(* CoDeSys 2.3.9.50 project: A_I_finale.pro *)
(* Libraries: STANDARD.LIB 5.6.98 12:03:02, Iecsfc.lib 12.5.98 12:03:00 *)

(* Task configuration *)
TASK Standard (PRIORITY := 0, INTERVAL := T#10ms);
	MAIN
END_TASK

(* POU MAIN, SFC *)
PROGRAM MAIN
VAR
	Presenza_pezzo								AT %IX0.0:BOOL;
	Colore_giostra								AT %IX0.1:BOOL;
	Pistone_avanti								AT %IX0.2:BOOL;
	Trapano_alto									AT %IX0.3:BOOL;
	Pistone_indietro								AT %IX0.4:BOOL;
	Trapano_basso								AT %IX0.5:BOOL;
	Fine_corsa_nastro								AT %IX0.6:BOOL;
	Tastatore_alto_altezza							AT %IX0.7:BOOL;


	Scarto_giostra_avanti_post_6					AT %IX1.0:BOOL;
	Scarto_giostra_indietro_post_6					AT %IX1.1:BOOL;
	Presenza_pezzo_baia							AT %IX1.2:BOOL;
	Tastatore_basso_altezza						AT %IX1.3:BOOL;
	Pennarello_alto								AT %IX1.4:BOOL;
	Pennarello_basso								AT %IX1.5:BOOL;
	Scarto_giostra_avanti_post_7					AT %IX1.6:BOOL;
	Scarto_giostra_indietro_post_7					AT %IX1.7:BOOL;


	Giostra_in_movimento							AT%IX2.0:BOOL;
	Sensore_vacuostato							AT%IX2.5:BOOL;
	Fine_corsa_braccio_magazzino					AT%IX2.6:BOOL;
	Presenza_pezzo_magazzino_B4					AT%IX2.7:BOOL;


	Pistone_indietro_1B2							AT%IX3.0:BOOL;
	Pistone_avanti_1B1							AT%IX3.1:BOOL;


	Fine_corsa_braccio_nastro						AT%IX4.1:BOOL;


(* ____ USCITE FISICHE____*)

	nastro  										AT %QX0.0:BOOL;
	pistone_giostra_post_6  						AT %QX0.1:BOOL;
	pistone_nastro		         						AT %QX0.2:BOOL;
	pennarello_down	     	    						AT %QX0.3:BOOL;
	movimento_giostra_1_posto  					AT %QX0.4:BOOL;
	pistone_giostra_post_7  						AT %QX0.5:BOOL;
	trapano_down								AT %QX0.6:BOOL;
	trapano_ON									AT %QX0.7:BOOL;

	tastatore_down								AT %QX1.0:BOOL;

	pistone_orizzontale							AT %QX2.1:BOOL;
	vacuostato									AT %QX2.2:BOOL;
	soffio_aria_ventosa							AT %QX2.3:BOOL;
	braccio_pneumatico_indietro					AT %QX2.4:BOOL;
	braccio_pneumatico_avanti						AT %QX2.5:BOOL;



(* ____ TIMER E CONTATORI IMPLEMENTATI____*)

(* ____ VARIABILI DI APPOGGIO VIRTUALI____*)

	attesa_magazzino: BOOL;
	pezzo_pronto_per_braccio: BOOL;
	pezzo_nel_braccio: BOOL;
	pezzo_pres: BOOL;
	riconoscimento_colore: BOOL;
	t_soffio: TON;
	attesa_secondi: BOOL;

	start:BOOL;
	emergenza:BOOL;
	accensione_pistone:BOOL;
	prova: tempo_3s;
	prova_2: tempo_3s;
	led_bottone: BOOL;
	lancio: BOOL;
	prov: TON;
	passaggio:BOOL;
	controllo_a_campione: CTU;
	pezzo_ok: BOOL;
	reset_cont: BOOL;
	contatore:BOOL;
END_VAR
VAR (* helpers for the ST form of the networks *)
	_p1 : BOOL;
	_p2 : BOOL;
END_VAR
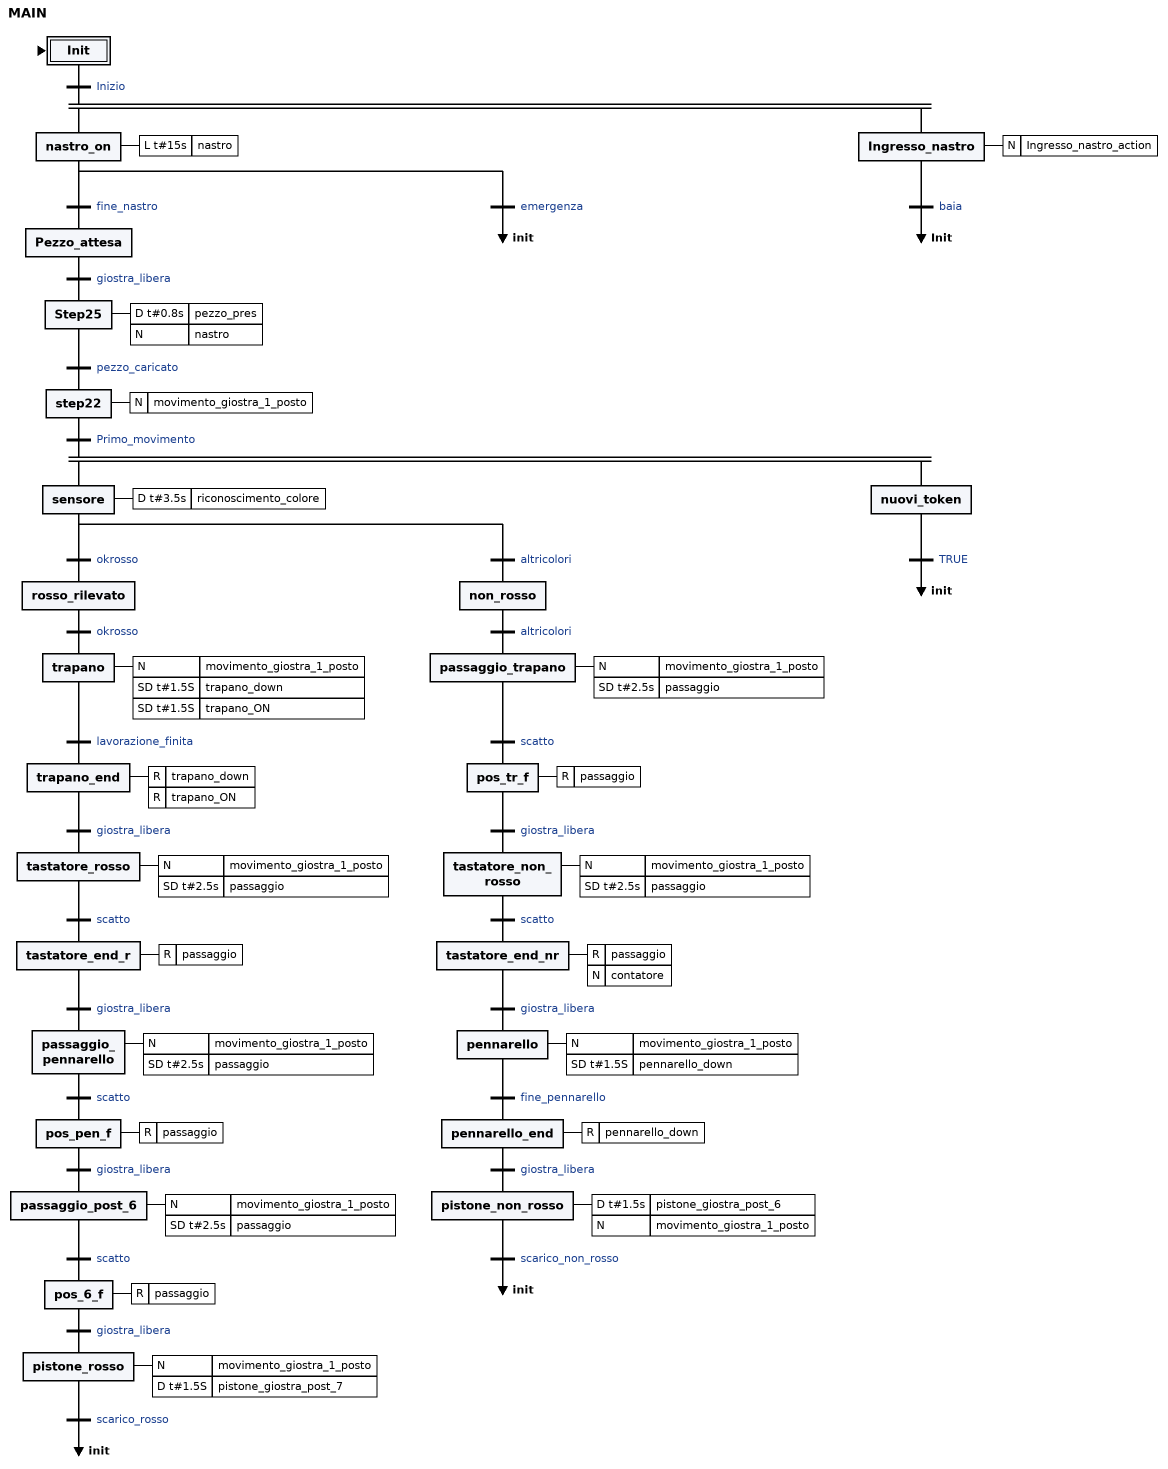
INITIAL_STEP Init:
END_STEP
TRANSITION FROM Init TO (nastro_on, Ingresso_nastro) := Inizio;
END_TRANSITION
STEP nastro_on:
	nastro(L, t#15s);
END_STEP
TRANSITION FROM nastro_on TO Pezzo_attesa := fine_nastro;
END_TRANSITION
TRANSITION FROM nastro_on TO init := emergenza;
END_TRANSITION
STEP Ingresso_nastro:
	Ingresso_nastro_action(N);
END_STEP
TRANSITION FROM Ingresso_nastro TO Init := baia;
END_TRANSITION
STEP Pezzo_attesa:
END_STEP
TRANSITION FROM Pezzo_attesa TO Step25 := giostra_libera;
END_TRANSITION
STEP Step25:
	pezzo_pres(D, t#0.8s);
	nastro(N);
END_STEP
TRANSITION FROM Step25 TO step22 := pezzo_caricato;
END_TRANSITION
STEP step22:
	movimento_giostra_1_posto(N);
END_STEP
TRANSITION FROM step22 TO (sensore, nuovi_token) := Primo_movimento;
END_TRANSITION
STEP sensore:
	riconoscimento_colore(D, t#3.5s);
END_STEP
TRANSITION FROM sensore TO rosso_rilevato := okrosso;
END_TRANSITION
TRANSITION FROM sensore TO non_rosso := altricolori;
END_TRANSITION
STEP nuovi_token:
END_STEP
TRANSITION FROM nuovi_token TO init := TRUE;
END_TRANSITION
STEP rosso_rilevato:
END_STEP
TRANSITION FROM rosso_rilevato TO trapano := okrosso;
END_TRANSITION
STEP trapano:
	movimento_giostra_1_posto(N);
	trapano_down(SD, t#1.5S);
	trapano_ON(SD, t#1.5S);
END_STEP
TRANSITION FROM trapano TO trapano_end := lavorazione_finita;
END_TRANSITION
STEP trapano_end:
	trapano_down(R);
	trapano_ON(R);
END_STEP
TRANSITION FROM trapano_end TO tastatore_rosso := giostra_libera;
END_TRANSITION
STEP tastatore_rosso:
	movimento_giostra_1_posto(N);
	passaggio(SD, t#2.5s);
END_STEP
TRANSITION FROM tastatore_rosso TO tastatore_end_r := scatto;
END_TRANSITION
STEP tastatore_end_r:
	passaggio(R);
END_STEP
TRANSITION FROM tastatore_end_r TO passaggio_pennarello := giostra_libera;
END_TRANSITION
STEP passaggio_pennarello:
	movimento_giostra_1_posto(N);
	passaggio(SD, t#2.5s);
END_STEP
TRANSITION FROM passaggio_pennarello TO pos_pen_f := scatto;
END_TRANSITION
STEP pos_pen_f:
	passaggio(R);
END_STEP
TRANSITION FROM pos_pen_f TO passaggio_post_6 := giostra_libera;
END_TRANSITION
STEP passaggio_post_6:
	movimento_giostra_1_posto(N);
	passaggio(SD, t#2.5s);
END_STEP
TRANSITION FROM passaggio_post_6 TO pos_6_f := scatto;
END_TRANSITION
STEP pos_6_f:
	passaggio(R);
END_STEP
TRANSITION FROM pos_6_f TO pistone_rosso := giostra_libera;
END_TRANSITION
STEP pistone_rosso:
	movimento_giostra_1_posto(N);
	pistone_giostra_post_7(D, t#1.5S);
END_STEP
TRANSITION FROM pistone_rosso TO init := scarico_rosso;
END_TRANSITION
STEP non_rosso:
END_STEP
TRANSITION FROM non_rosso TO passaggio_trapano := altricolori;
END_TRANSITION
STEP passaggio_trapano:
	movimento_giostra_1_posto(N);
	passaggio(SD, t#2.5s);
END_STEP
TRANSITION FROM passaggio_trapano TO pos_tr_f := scatto;
END_TRANSITION
STEP pos_tr_f:
	passaggio(R);
END_STEP
TRANSITION FROM pos_tr_f TO tastatore_non_rosso := giostra_libera;
END_TRANSITION
STEP tastatore_non_rosso:
	movimento_giostra_1_posto(N);
	passaggio(SD, t#2.5s);
END_STEP
TRANSITION FROM tastatore_non_rosso TO tastatore_end_nr := scatto;
END_TRANSITION
STEP tastatore_end_nr:
	passaggio(R);
	contatore(N);
END_STEP
TRANSITION FROM tastatore_end_nr TO pennarello := giostra_libera;
END_TRANSITION
STEP pennarello:
	movimento_giostra_1_posto(N);
	pennarello_down(SD, t#1.5S);
END_STEP
TRANSITION FROM pennarello TO pennarello_end := fine_pennarello;
END_TRANSITION
STEP pennarello_end:
	pennarello_down(R);
END_STEP
TRANSITION FROM pennarello_end TO pistone_non_rosso := giostra_libera;
END_TRANSITION
STEP pistone_non_rosso:
	pistone_giostra_post_6(D, t#1.5s);
	movimento_giostra_1_posto(N);
END_STEP
TRANSITION FROM pistone_non_rosso TO init := scarico_non_rosso;
END_TRANSITION

ACTION Ingresso_nastro_action:
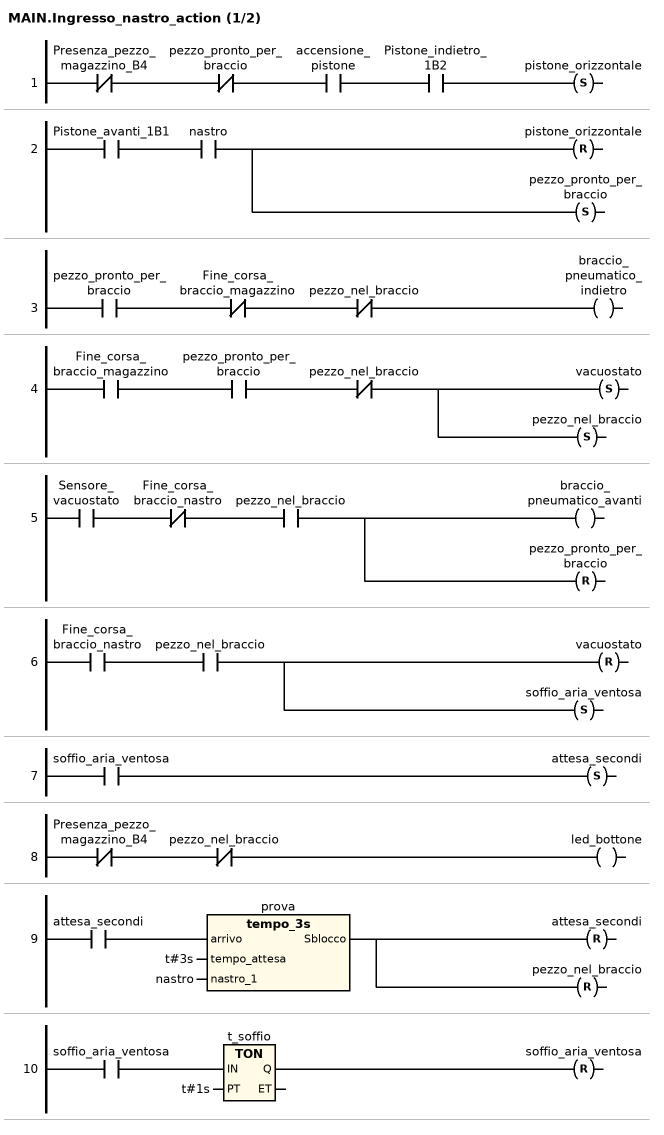
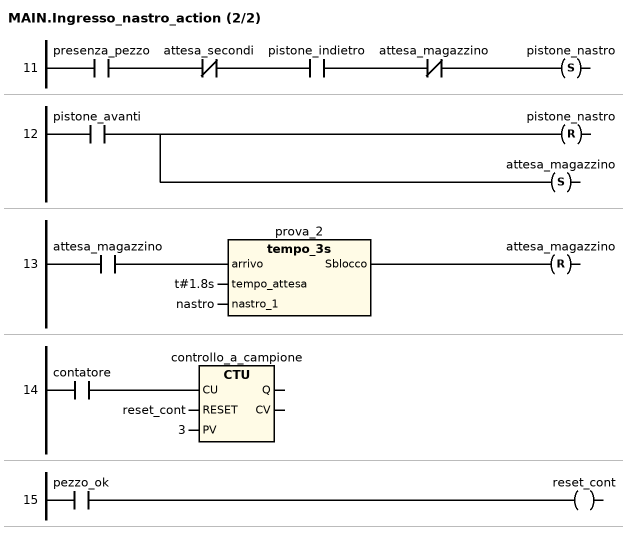
_LD_ (* Ladder Diagram *)
NETWORK 1
	[/Presenza_pezzo_magazzino_B4] - [/pezzo_pronto_per_braccio] - [accensione_pistone] - [Pistone_indietro_1B2] --- (S pistone_orizzontale)
NETWORK 2
	[Pistone_avanti_1B1] - [nastro] --- (R pistone_orizzontale) (S pezzo_pronto_per_braccio)
NETWORK 3
	[pezzo_pronto_per_braccio] - [/Fine_corsa_braccio_magazzino] - [/pezzo_nel_braccio] --- (braccio_pneumatico_indietro)
NETWORK 4
	[Fine_corsa_braccio_magazzino] - [pezzo_pronto_per_braccio] - [/pezzo_nel_braccio] --- (S vacuostato) (S pezzo_nel_braccio)
NETWORK 5
	[Sensore_vacuostato] - [/Fine_corsa_braccio_nastro] - [pezzo_nel_braccio] --- (braccio_pneumatico_avanti) (R pezzo_pronto_per_braccio)
NETWORK 6
	[Fine_corsa_braccio_nastro] - [pezzo_nel_braccio] --- (R vacuostato) (S soffio_aria_ventosa)
NETWORK 7
	[soffio_aria_ventosa] --- (S attesa_secondi)
NETWORK 8
	[/Presenza_pezzo_magazzino_B4] - [/pezzo_nel_braccio] --- (led_bottone)
NETWORK 9
	[attesa_secondi] - prova:tempo_3s(arrivo: *, tempo_attesa: t#3s, nastro_1: nastro) --- (R attesa_secondi) (R pezzo_nel_braccio)
NETWORK 10
	[soffio_aria_ventosa] - t_soffio:TON(IN: *, PT: t#1s) --- (R soffio_aria_ventosa)
NETWORK 11
	[presenza_pezzo] - [/attesa_secondi] - [pistone_indietro] - [/attesa_magazzino] --- (S pistone_nastro)
NETWORK 12
	[pistone_avanti] --- (R pistone_nastro) (S attesa_magazzino)
NETWORK 13
	[attesa_magazzino] - prova_2:tempo_3s(arrivo: *, tempo_attesa: t#1.8s, nastro_1: nastro) --- (R attesa_magazzino)
NETWORK 14
	[contatore] - controllo_a_campione:CTU(CU: *, RESET: reset_cont, PV: 3)
NETWORK 15
	[pezzo_ok] --- (reset_cont)
_END_LD_
(* the same logic as Structured Text *)
(* Network 1 *)
IF NOT Presenza_pezzo_magazzino_B4 AND NOT pezzo_pronto_per_braccio AND accensione_pistone AND Pistone_indietro_1B2 THEN pistone_orizzontale := TRUE; END_IF;
(* Network 2 *)
IF Pistone_avanti_1B1 AND nastro THEN pistone_orizzontale := FALSE; pezzo_pronto_per_braccio := TRUE; END_IF;
(* Network 3 *)
braccio_pneumatico_indietro := pezzo_pronto_per_braccio AND NOT Fine_corsa_braccio_magazzino AND NOT pezzo_nel_braccio;
(* Network 4 *)
_p1 := Fine_corsa_braccio_magazzino AND pezzo_pronto_per_braccio AND NOT pezzo_nel_braccio;
IF _p1 THEN vacuostato := TRUE; pezzo_nel_braccio := TRUE; END_IF;
(* Network 5 *)
braccio_pneumatico_avanti := Sensore_vacuostato AND NOT Fine_corsa_braccio_nastro AND pezzo_nel_braccio;
IF braccio_pneumatico_avanti THEN pezzo_pronto_per_braccio := FALSE; END_IF;
(* Network 6 *)
_p2 := Fine_corsa_braccio_nastro AND pezzo_nel_braccio;
IF _p2 THEN vacuostato := FALSE; soffio_aria_ventosa := TRUE; END_IF;
(* Network 7 *)
IF soffio_aria_ventosa THEN attesa_secondi := TRUE; END_IF;
(* Network 8 *)
led_bottone := NOT Presenza_pezzo_magazzino_B4 AND NOT pezzo_nel_braccio;
(* Network 9 *)
prova(arrivo := attesa_secondi, tempo_attesa := t#3s, nastro_1 := nastro);
IF prova.Sblocco THEN attesa_secondi := FALSE; pezzo_nel_braccio := FALSE; END_IF;
(* Network 10 *)
t_soffio(IN := soffio_aria_ventosa, PT := t#1s);
IF t_soffio.Q THEN soffio_aria_ventosa := FALSE; END_IF;
(* Network 11 *)
IF presenza_pezzo AND NOT attesa_secondi AND pistone_indietro AND NOT attesa_magazzino THEN pistone_nastro := TRUE; END_IF;
(* Network 12 *)
IF pistone_avanti THEN pistone_nastro := FALSE; attesa_magazzino := TRUE; END_IF;
(* Network 13 *)
prova_2(arrivo := attesa_magazzino, tempo_attesa := t#1.8s, nastro_1 := nastro);
IF prova_2.Sblocco THEN attesa_magazzino := FALSE; END_IF;
(* Network 14 *)
controllo_a_campione(CU := contatore, RESET := reset_cont, PV := 3);
(* Network 15 *)
reset_cont := pezzo_ok;
END_ACTION

TRANSITION Inizio:
_LD_ (* Ladder Diagram *)
NETWORK 1
	[/Presenza_pezzo_baia] - [/emergenza] - [start]
_END_LD_
(* the same logic as Structured Text *)
(* Network 1 *)
Inizio := NOT Presenza_pezzo_baia AND NOT emergenza AND start;
END_TRANSITION

TRANSITION baia:
_LD_ (* Ladder Diagram *)
NETWORK 1
	{ [Presenza_pezzo_baia] | [emergenza] }
_END_LD_
(* the same logic as Structured Text *)
(* Network 1 *)
baia := Presenza_pezzo_baia OR emergenza;
END_TRANSITION

TRANSITION fine_nastro:
_LD_ (* Ladder Diagram *)
NETWORK 1
	[/Fine_corsa_nastro]
_END_LD_
(* the same logic as Structured Text *)
(* Network 1 *)
fine_nastro := NOT Fine_corsa_nastro;
END_TRANSITION

TRANSITION giostra_libera:
_LD_ (* Ladder Diagram *)
NETWORK 1
	[/Presenza_pezzo_baia] - [Trapano_alto] - [TRUE] - [Pennarello_alto] - [Scarto_giostra_indietro_post_6] - [Scarto_giostra_indietro_post_7] - [/Giostra_in_movimento] - [/SENSORE.x] - [/emergenza] - [/passaggio] - [/controllo_a_campione.Q]
_END_LD_
(* the same logic as Structured Text *)
(* Network 1 *)
giostra_libera := NOT Presenza_pezzo_baia AND Trapano_alto AND TRUE AND Pennarello_alto AND Scarto_giostra_indietro_post_6 AND Scarto_giostra_indietro_post_7 AND NOT Giostra_in_movimento AND NOT SENSORE.x AND NOT emergenza AND NOT passaggio AND NOT controllo_a_campione.Q;
END_TRANSITION

TRANSITION pezzo_caricato:
_LD_ (* Ladder Diagram *)
NETWORK 1
	[pezzo_pres]
_END_LD_
(* the same logic as Structured Text *)
(* Network 1 *)
pezzo_caricato := pezzo_pres;
END_TRANSITION

TRANSITION Primo_movimento:
_LD_ (* Ladder Diagram *)
NETWORK 1
	[movimento_giostra_1_posto]
_END_LD_
(* the same logic as Structured Text *)
(* Network 1 *)
Primo_movimento := movimento_giostra_1_posto;
END_TRANSITION

TRANSITION okrosso:
_LD_ (* Ladder Diagram *)
NETWORK 1
	[riconoscimento_colore] - [Colore_giostra]
_END_LD_
(* the same logic as Structured Text *)
(* Network 1 *)
okrosso := riconoscimento_colore AND Colore_giostra;
END_TRANSITION

TRANSITION okrosso:
_LD_ (* Ladder Diagram *)
NETWORK 1
	[/Presenza_pezzo_baia] - [Trapano_alto] - [TRUE] - [Pennarello_alto] - [Scarto_giostra_indietro_post_6] - [Scarto_giostra_indietro_post_7] - [/Giostra_in_movimento] - [/PEZZO_ATTESA.x] - [/STEP25.x] - [/emergenza] - [/passaggio] - [/controllo_a_campione.Q]
_END_LD_
(* the same logic as Structured Text *)
(* Network 1 *)
okrosso := NOT Presenza_pezzo_baia AND Trapano_alto AND TRUE AND Pennarello_alto AND Scarto_giostra_indietro_post_6 AND Scarto_giostra_indietro_post_7 AND NOT Giostra_in_movimento AND NOT PEZZO_ATTESA.x AND NOT STEP25.x AND NOT emergenza AND NOT passaggio AND NOT controllo_a_campione.Q;
END_TRANSITION

TRANSITION lavorazione_finita:
_LD_ (* Ladder Diagram *)
NETWORK 1
	[Trapano_basso]
_END_LD_
(* the same logic as Structured Text *)
(* Network 1 *)
lavorazione_finita := Trapano_basso;
END_TRANSITION

TRANSITION giostra_libera:
_LD_ (* Ladder Diagram *)
NETWORK 1
	[/Presenza_pezzo_baia] - [Trapano_alto] - [TRUE] - [Pennarello_alto] - [Scarto_giostra_indietro_post_6] - [Scarto_giostra_indietro_post_7] - [/Giostra_in_movimento] - [/PEZZO_ATTESA.x] - [/STEP22.x] - [/STEP25.x] - [/emergenza] - [/passaggio] - [/controllo_a_campione.Q]
_END_LD_
(* the same logic as Structured Text *)
(* Network 1 *)
giostra_libera := NOT Presenza_pezzo_baia AND Trapano_alto AND TRUE AND Pennarello_alto AND Scarto_giostra_indietro_post_6 AND Scarto_giostra_indietro_post_7 AND NOT Giostra_in_movimento AND NOT PEZZO_ATTESA.x AND NOT STEP22.x AND NOT STEP25.x AND NOT emergenza AND NOT passaggio AND NOT controllo_a_campione.Q;
END_TRANSITION

TRANSITION scatto:
_LD_ (* Ladder Diagram *)
NETWORK 1
	[passaggio]
_END_LD_
(* the same logic as Structured Text *)
(* Network 1 *)
scatto := passaggio;
END_TRANSITION

TRANSITION giostra_libera:
_LD_ (* Ladder Diagram *)
NETWORK 1
	[/Presenza_pezzo_baia] - [Trapano_alto] - [TRUE] - [Pennarello_alto] - [Scarto_giostra_indietro_post_6] - [Scarto_giostra_indietro_post_7] - [/Giostra_in_movimento] - [/PEZZO_ATTESA.x] - [/STEP22.x] - [/STEP25.x] - [/emergenza] - [/passaggio] - [/controllo_a_campione.Q]
_END_LD_
(* the same logic as Structured Text *)
(* Network 1 *)
giostra_libera := NOT Presenza_pezzo_baia AND Trapano_alto AND TRUE AND Pennarello_alto AND Scarto_giostra_indietro_post_6 AND Scarto_giostra_indietro_post_7 AND NOT Giostra_in_movimento AND NOT PEZZO_ATTESA.x AND NOT STEP22.x AND NOT STEP25.x AND NOT emergenza AND NOT passaggio AND NOT controllo_a_campione.Q;
END_TRANSITION

TRANSITION scatto:
_LD_ (* Ladder Diagram *)
NETWORK 1
	[passaggio]
_END_LD_
(* the same logic as Structured Text *)
(* Network 1 *)
scatto := passaggio;
END_TRANSITION

TRANSITION giostra_libera:
_LD_ (* Ladder Diagram *)
NETWORK 1
	[/Presenza_pezzo_baia] - [Trapano_alto] - [TRUE] - [Pennarello_alto] - [Scarto_giostra_indietro_post_6] - [Scarto_giostra_indietro_post_7] - [/Giostra_in_movimento] - [/PEZZO_ATTESA.x] - [/STEP22.x] - [/STEP25.x] - [/emergenza] - [/passaggio] - [/controllo_a_campione.Q]
_END_LD_
(* the same logic as Structured Text *)
(* Network 1 *)
giostra_libera := NOT Presenza_pezzo_baia AND Trapano_alto AND TRUE AND Pennarello_alto AND Scarto_giostra_indietro_post_6 AND Scarto_giostra_indietro_post_7 AND NOT Giostra_in_movimento AND NOT PEZZO_ATTESA.x AND NOT STEP22.x AND NOT STEP25.x AND NOT emergenza AND NOT passaggio AND NOT controllo_a_campione.Q;
END_TRANSITION

TRANSITION scatto:
_LD_ (* Ladder Diagram *)
NETWORK 1
	[passaggio]
_END_LD_
(* the same logic as Structured Text *)
(* Network 1 *)
scatto := passaggio;
END_TRANSITION

TRANSITION giostra_libera:
_LD_ (* Ladder Diagram *)
NETWORK 1
	[/Presenza_pezzo_baia] - [Trapano_alto] - [TRUE] - [Pennarello_alto] - [Scarto_giostra_indietro_post_6] - [Scarto_giostra_indietro_post_7] - [/Giostra_in_movimento] - [/PEZZO_ATTESA.x] - [/STEP22.x] - [/STEP25.x] - [/emergenza] - [/passaggio] - [/controllo_a_campione.Q]
_END_LD_
(* the same logic as Structured Text *)
(* Network 1 *)
giostra_libera := NOT Presenza_pezzo_baia AND Trapano_alto AND TRUE AND Pennarello_alto AND Scarto_giostra_indietro_post_6 AND Scarto_giostra_indietro_post_7 AND NOT Giostra_in_movimento AND NOT PEZZO_ATTESA.x AND NOT STEP22.x AND NOT STEP25.x AND NOT emergenza AND NOT passaggio AND NOT controllo_a_campione.Q;
END_TRANSITION

TRANSITION scarico_rosso:
_LD_ (* Ladder Diagram *)
NETWORK 1
	[/Presenza_pezzo_baia] - [Scarto_giostra_avanti_post_7]
_END_LD_
(* the same logic as Structured Text *)
(* Network 1 *)
scarico_rosso := NOT Presenza_pezzo_baia AND Scarto_giostra_avanti_post_7;
END_TRANSITION

TRANSITION altricolori:
_LD_ (* Ladder Diagram *)
NETWORK 1
	[riconoscimento_colore] - [/Colore_giostra]
_END_LD_
(* the same logic as Structured Text *)
(* Network 1 *)
altricolori := riconoscimento_colore AND NOT Colore_giostra;
END_TRANSITION

TRANSITION altricolori:
_LD_ (* Ladder Diagram *)
NETWORK 1
	[/Presenza_pezzo_baia] - [Trapano_alto] - [TRUE] - [Pennarello_alto] - [Scarto_giostra_indietro_post_6] - [Scarto_giostra_indietro_post_7] - [/Giostra_in_movimento] - [/PEZZO_ATTESA.x] - [/STEP25.x] - [/emergenza] - [/passaggio] - [/controllo_a_campione.Q]
_END_LD_
(* the same logic as Structured Text *)
(* Network 1 *)
altricolori := NOT Presenza_pezzo_baia AND Trapano_alto AND TRUE AND Pennarello_alto AND Scarto_giostra_indietro_post_6 AND Scarto_giostra_indietro_post_7 AND NOT Giostra_in_movimento AND NOT PEZZO_ATTESA.x AND NOT STEP25.x AND NOT emergenza AND NOT passaggio AND NOT controllo_a_campione.Q;
END_TRANSITION

TRANSITION scatto:
_LD_ (* Ladder Diagram *)
NETWORK 1
	[passaggio]
_END_LD_
(* the same logic as Structured Text *)
(* Network 1 *)
scatto := passaggio;
END_TRANSITION

TRANSITION giostra_libera:
_LD_ (* Ladder Diagram *)
NETWORK 1
	[/Presenza_pezzo_baia] - [Trapano_alto] - [TRUE] - [Pennarello_alto] - [Scarto_giostra_indietro_post_6] - [Scarto_giostra_indietro_post_7] - [/Giostra_in_movimento] - [/PEZZO_ATTESA.x] - [/STEP22.x] - [/STEP25.x] - [/emergenza] - [/passaggio] - [/controllo_a_campione.Q]
_END_LD_
(* the same logic as Structured Text *)
(* Network 1 *)
giostra_libera := NOT Presenza_pezzo_baia AND Trapano_alto AND TRUE AND Pennarello_alto AND Scarto_giostra_indietro_post_6 AND Scarto_giostra_indietro_post_7 AND NOT Giostra_in_movimento AND NOT PEZZO_ATTESA.x AND NOT STEP22.x AND NOT STEP25.x AND NOT emergenza AND NOT passaggio AND NOT controllo_a_campione.Q;
END_TRANSITION

TRANSITION scatto:
_LD_ (* Ladder Diagram *)
NETWORK 1
	[passaggio]
_END_LD_
(* the same logic as Structured Text *)
(* Network 1 *)
scatto := passaggio;
END_TRANSITION

TRANSITION giostra_libera:
_LD_ (* Ladder Diagram *)
NETWORK 1
	[/Presenza_pezzo_baia] - [Trapano_alto] - [TRUE] - [Pennarello_alto] - [Scarto_giostra_indietro_post_6] - [Scarto_giostra_indietro_post_7] - [/Giostra_in_movimento] - [/STEP22.x] - [/STEP25.x] - [/emergenza] - [/passaggio] - { [/controllo_a_campione.Q] | [controllo_a_campione.Q] - [pezzo_ok] } - [/PEZZO_ATTESA.x]
_END_LD_
(* the same logic as Structured Text *)
(* Network 1 *)
giostra_libera := NOT Presenza_pezzo_baia AND Trapano_alto AND TRUE AND Pennarello_alto AND Scarto_giostra_indietro_post_6 AND Scarto_giostra_indietro_post_7 AND NOT Giostra_in_movimento AND NOT STEP22.x AND NOT STEP25.x AND NOT emergenza AND NOT passaggio AND (NOT controllo_a_campione.Q OR controllo_a_campione.Q AND pezzo_ok) AND NOT PEZZO_ATTESA.x;
END_TRANSITION

TRANSITION fine_pennarello:
_LD_ (* Ladder Diagram *)
NETWORK 1
	[Pennarello_basso]
_END_LD_
(* the same logic as Structured Text *)
(* Network 1 *)
fine_pennarello := Pennarello_basso;
END_TRANSITION

TRANSITION giostra_libera:
_LD_ (* Ladder Diagram *)
NETWORK 1
	[/Presenza_pezzo_baia] - [Trapano_alto] - [TRUE] - [Pennarello_alto] - [Scarto_giostra_indietro_post_6] - [Scarto_giostra_indietro_post_7] - [/Giostra_in_movimento] - [/PEZZO_ATTESA.x] - [/STEP22.x] - [/STEP25.x] - [/emergenza] - [/passaggio] - [/controllo_a_campione.Q]
_END_LD_
(* the same logic as Structured Text *)
(* Network 1 *)
giostra_libera := NOT Presenza_pezzo_baia AND Trapano_alto AND TRUE AND Pennarello_alto AND Scarto_giostra_indietro_post_6 AND Scarto_giostra_indietro_post_7 AND NOT Giostra_in_movimento AND NOT PEZZO_ATTESA.x AND NOT STEP22.x AND NOT STEP25.x AND NOT emergenza AND NOT passaggio AND NOT controllo_a_campione.Q;
END_TRANSITION

TRANSITION scarico_non_rosso:
_LD_ (* Ladder Diagram *)
NETWORK 1
	[/Presenza_pezzo_baia] - [Scarto_giostra_avanti_post_6]
_END_LD_
(* the same logic as Structured Text *)
(* Network 1 *)
scarico_non_rosso := NOT Presenza_pezzo_baia AND Scarto_giostra_avanti_post_6;
END_TRANSITION
END_PROGRAM

(* POU tempo_3s, ST *)
FUNCTION_BLOCK tempo_3s
VAR_INPUT
	arrivo: BOOL;
	tempo_attesa: TIME;
  	nastro_1: BOOL;
END_VAR
VAR_OUTPUT
	Sblocco:BOOL := FALSE;
END_VAR
VAR
	MyTimer: TON;
	TotalET: TIME:= T#0s;
	prova: TIME :=T#0s;
END_VAR
	MyTimer(IN := (nastro_1 AND arrivo), PT := tempo_attesa);
	IF nastro_1 = TRUE
		THEN
		prova := MyTimer.ET;
	END_IF

	IF nastro_1 = FALSE
	THEN
	TotalET := TotalET + prova;
	prova := t#0s;
	END_IF

	IF  ( (TotalET + prova) >= tempo_attesa)
		THEN
		sblocco := TRUE;
		TotalET := t#0s;
		prova := t#0s;
	ELSE
		sblocco := FALSE;
	END_IF
END_FUNCTION_BLOCK

(* Visualisation PULSANTI
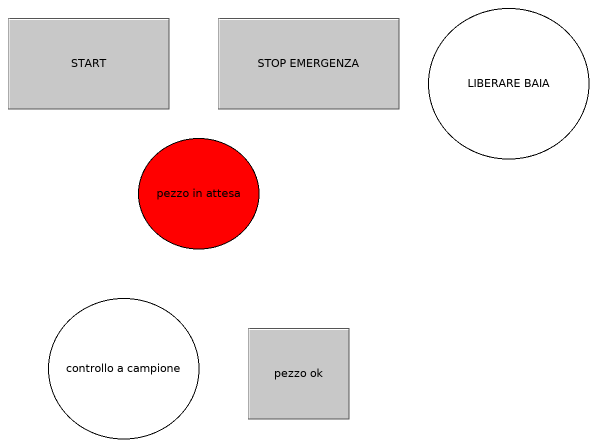
button at (20,20)-(181,111): text "START"; toggles MAIN.start
button at (230,20)-(411,111): text "STOP EMERGENZA"; toggles MAIN.emergenza
ellipse at (150,140)-(271,251): text "pezzo in attesa"; alarm colour if MAIN.led_bottone
ellipse at (440,10)-(601,161): text "LIBERARE BAIA"; alarm colour if MAIN.Presenza_pezzo_baia
ellipse at (60,300)-(211,441): text "controllo a campione"; alarm colour if MAIN.controllo_a_campione.Q
button at (260,330)-(361,421): text "pezzo ok"; taps MAIN.pezzo_ok
1 elements of other kinds (tables, trends, ...) not read
*)
